// TIA Portal V20 export
FUNCTION_BLOCK "RealFbName"   // FB2, LAD
   VAR RETAIN
      IO { S7_SetPoint := 'True'} : "TypeDOL";
   END_VAR
   VAR
      FaultTripTimer2 { S7_SetPoint := 'True'} : TON_TIME;
   END_VAR
   VAR_TEMP
      "Time" : Real;
   END_VAR
   // IO.InHand := FALSE;
BEGIN
END_FUNCTION_BLOCK
